TYPE ST_P50A_Haupt_OUT :
STRUCT
	bLedDoorOpn			: BOOL;	// Schutztüren Entriegeln, LDT-WH, 1DI-NO, 1DO, BMK: +P50A-21SJ5
 	bLedVorwHaerten		: BOOL;	// Vorwahl Härte-Generator, LDT-WH, 1DI-NO, 1DO, BMK: +P50A-22SJ1
	bLedVorwAnlassen	: BOOL;	// Vorwahl Anlass-Generator, LDT-WH, 1DI-NO, 1DO, BMK: +P50A-22SJ2
	bLedPolieren		: BOOL;	// Polierstation Start/Stopp, LDT-WH, 1DI-NO, 1DO, BMK: +P50A-22SJ3
	bLedSpS1			: BOOL;	// Spindel S1 Start/Stopp, LDT-WH, 1DI-NO, 1DO, BMK: +P50A-22SJ5
	bLedSpS2			: BOOL;	// Spindel S2 Start/Stopp, LDT-WH, 1DI-NO, 1DO, BMK: +P50A-23SJ1
	bLedSpS3			: BOOL;	// Spindel S3 Start/Stopp, LDT-WH, 1DI-NO, 1DO, BMK: +P50A-23SJ5
	bLedAutoOn			: BOOL;	// Automatik Ein, LDT-GN, 1DI-NO, 1DO, BMK: +P50A-21SJ2

	bLedDoorCls			: BOOL;	// Schutztüren Verriegeln, LDT-WH, 1DI-NO, 1DO, BMK: +P50A-21SJ6
	bLedHaerteGen		: BOOL;	// Härte-Generator Status, LM-GN, 1DO, BMK: +P50A-32PF2
	bLedAnlassGen		: BOOL;	// Anlss-Generator Status, LM-GN, 1DO, BMK: +P50A-32PF4
	bLedZustPolieren	: BOOL;	// Polierstation Zustellung, LDT-WH, 1DI-NO, 1DO, BMK: +P50A-22SJ4
	bLedZustS1			: BOOL;	// Spindel S1 Zustellung, LDT-WH, 1DI-NO, 1DO, BMK: +P50A-22SJ6
	bLedZustS2			: BOOL;	// Spindel S2 Zustellung, LDT-WH, 1DI-NO, 1DO, BMK: +P50A-23SJ2
	bLedZustS3			: BOOL;	// Spindel S3 Zustellung, LDT-WH, 1DI-NO, 1DO, BMK: +P50A-23SJ6	

	bLedEnAutoKorrS1	: BOOL;	// Spindel S1 Autokorrektur Ein/Aus, LDT-WH, 1DI-NO, 1DO, BMK: +P50A-22SJ7
	bLedEnAutoKorrS2	: BOOL;	// Spindel S2 Autokorrektur Ein/Aus, LDT-WH, 1DI-NO, 1DO, BMK: +P50A-23SJ3
	bLedEnAutoKorrS3	: BOOL;	// Spindel S3 Autokorrektur Ein/Aus, LDT-WH, 1DI-NO, 1DO, BMK: +P50A-23SJ7
	bLedQuit			: BOOL;	// Not-Halt Quittieren, LDT-BU, 1DI-NO, 1DO, BMK: +P50A-21SJ1

END_STRUCT
END_TYPE

(* stored: Version 1.1.0.1, ProductVersion 3.1.4024.12
   DUT ST_P50A_Haupt_OUT: Id {601e7d79-310b-4064-834f-27e18838fbc3} *)
